FUNCTION_BLOCK GeneratedTest EXTENDS TcUnit.FB_TestSuite

END_FUNCTION_BLOCK

(* stored: Version 1.1.0.1, ProductVersion 3.1.4024.9
   POU GeneratedTest: Id {8a002d40-1b8b-4a36-917f-04dd149a7db3}, SpecialFunc None *)
